{attribute 'GeneratedUsingTerminal: IL2301-B110-0016'}
{attribute addProperty BoxType "IL2301-B110-0016"}
{attribute addProperty Id "Term_21KL_D4CFBC220Term_392_Ix1000KL_8EF4D3E90"}
{attribute addProperty CRC "4284580109"}
{attribute addProperty Size "0"}
TYPE A_0021_IL2301_B110_0016_FF61810D EXTENDS IL2301_A2FCADE7 :
STRUCT
	{attribute addProperty Name "Term_21"}
	Term_21 : KL_D4CFBC22;
	{attribute addProperty Name "Term_392_Ix1000"}
	Term_392_Ix1000 : KL_8EF4D3E9;
END_STRUCT
END_TYPE

(* stored: Version 1.2.0.0, ProductVersion 3.1.4024.9
   DUT A_0021_IL2301_B110_0016_FF61810D: Id {0ca22d70-035b-419d-956f-492504a7212c} *)
